KUKA KRL program: Prelaunch.src

&ACCESS RVP
&REL 1
&PARAM TEMPLATE = C:\KRC\Roboter\Template\vorgabe
&PARAM EDITMASK = *
DEF Prelaunch ( )
EXT BAS (BAS_COMMAND :IN,REAL :IN )


; GLOBAL INTERRUPT DECL 3 WHEN $STOPMESS==TRUE DO IR_STOPM ( )
; INTERRUPT ON 3

;FOLD Initialise and set default speed
BAS (#INITMOV,0)
BAS (#VEL_PTP,100)
BAS (#ACC_PTP,20)
$VEL.CP=0.2
BAS (#TOOL,0)
BAS (#BASE,0)
;ENDFOLD

;;FOLD STARTPOS
;$BWDSTART = FALSE
;PDAT_ACT = PDEFAULT
;BAS(#PTP_DAT)
;FDAT_ACT = {TOOL_NO 0,BASE_NO 0,IPO_FRAME #BASE}
;BAS(#FRAMES)
;;ENDFOLD

$ADVANCE = 5

;FOLD ---- Quickly skip BCO ----
; PTP $AXIS_ACT
;ENDFOLD

;FOLD ---- GO HOME ----
; PTP {A1 0.000, A2 -90.000, A3 90.000, A4 0.000, A5 0.000, A6 0.000, E1 0, E2 0, E3 0, E4 0, E5 0, E6 0}
;ENDFOLD


; Program generated by RoboDK v5.9.5 for KUKA KR 150 L120/2 on 12/01/2026 20:41:23
; Using nominal kinematics.
; ---- Setting reference (Base) ----
; BASE_DATA[2] = {FRAME: X -1800.000,Y 1305.450,Z 600.000,A -90.000,B 0.000,C 0.000}
$BASE = {FRAME: X -1800.000,Y 1305.450,Z 600.000,A -90.000,B 0.000,C 0.000}
; $BASE = BASE_DATA[2]
; --------------------------
; ---- Setting tool (TCP) ----
$TOOL = {FRAME: X 0.000,Y 0.000,Z 200.000,A 0.000,B 0.000,C 0.000}
; --------------------------
PTP {A1 -27.73790,A2 -54.67830,A3 100.89100,A4 -171.55600,A5 46.52490,A6 174.16800}
PTP {A1 -142.84300,A2 -73.92970,A3 132.07000,A4 -280.67200,A5 93.59510,A6 206.12700}
END
